TYPE BandPassFilterStruct :
STRUCT
	G1_a0 : REAL;
	G1_a1 : REAL;
	G1_a2 : REAL;

	G1_b0 : REAL;
	
	output : REAL;
	error1 : REAL;
	error2 : REAL;
	output1 : REAL;
	output2 : REAL;

END_STRUCT
END_TYPE

(* stored: Version 1.1.0.1, ProductVersion 3.1.4024.4
   DUT BandPassFilterStruct: Id {92776ef2-d8ed-4dda-a587-ffa1810c050b} *)
